(* IEC 61131-3 sources: generating_plc_code_with_llms/Code#1/ChatGPT_4/first run, 21 files *)

(* ---- 14.st ---- *)
// 41.85s
// 4
FUNCTION FC1001 : BOOL
VAR_INPUT
    MeasuredValue : REAL;  // The current measured value from the sensor
    SwitchValue   : REAL;  // The predetermined switch value
    Hysteresis    : REAL;  // The hysteresis in percentage of the switch value
END_VAR

VAR
    UpperLimit : REAL;
    LowerLimit : REAL;
END_VAR

// Calculate the upper and lower limits based on the hysteresis
UpperLimit := SwitchValue + (SwitchValue * Hysteresis / 100);
LowerLimit := SwitchValue - (SwitchValue * Hysteresis / 100);

// Logic to turn the output on or off based on the measured value and hysteresis
IF MeasuredValue > UpperLimit THEN
    FC1001 := TRUE;  // Turn on the output
ELSIF MeasuredValue < LowerLimit THEN
    FC1001 := FALSE; // Turn off the output
// If the value is within the hysteresis range, keep the output as is
END_IF

(* ---- 15.st ---- *)
// 58.63s
// 3
FUNCTION FC1002
VAR_INPUT
    SensorDetected : BOOL;  // TRUE if the ultrasonic sensor detects something
    E_A            : BOOL;  // The switch to turn the monitoring system on/off
END_VAR

VAR_OUTPUT
    P_HU           : BOOL;  // The horn for acoustic warning
    P_AL           : BOOL;  // The alarm
    P1             : BOOL;  // Indicator for monitoring system status
END_VAR

VAR
    DetectionTimer : TON;   // Timer for detection duration
END_VAR

// Turn on the monitoring system and indicate status
IF E_A THEN
    P1 := TRUE;
ELSE
    P1 := FALSE;
    P_HU := FALSE;  // Turn off horn when system is turned off
    P_AL := FALSE;  // Turn off alarm when system is turned off
END_IF

// Handling sensor detection
IF SensorDetected THEN
    IF NOT DetectionTimer.IN THEN
        DetectionTimer(IN := TRUE, PT := T#3s);  // Start timer when detection begins
    END_IF
    IF DetectionTimer.Q THEN
        P_HU := FALSE;  // Turn off horn after 3 seconds
        P_AL := TRUE;   // Turn on alarm after 3 seconds
    ELSE
        P_HU := TRUE;   // Turn on horn when detection is within 3 seconds
    END_IF
ELSE
    DetectionTimer(IN := FALSE);  // Reset timer when no detection
    P_HU := FALSE;                // Turn off horn if nothing is detected
    // Keep alarm on if it was already triggered, unless the system is turned off
END_IF

(* ---- 18.st ---- *)
// 37.97s
// 4
FUNCTION FC1003 : REAL
VAR_INPUT
    InputValue : REAL;    // The value from the sensor (0 to 255 in your case)
    IN_MIN     : REAL;    // Lower limit of the input range
    IN_MAX     : REAL;    // Upper limit of the input range
    OUT_MIN    : REAL;    // Lower limit of the output range (e.g., -20C)
    OUT_MAX    : REAL;    // Upper limit of the output range (e.g., 40C)
END_VAR

BEGIN
    // Linearly map the input value from its range to the output range
    FC1003 := OUT_MIN + (InputValue - IN_MIN) * (OUT_MAX - OUT_MIN) / (IN_MAX - IN_MIN);
END_FUNCTION

(* ---- 2.st ---- *)
//30.22s
//2
(* Function to calculate factorial *)
FUNCTION Factorial : LINT
VAR_INPUT
    n : UINT; (* non-negative integer *)
END_VAR
VAR
    result : LINT := 1; (* Initialize result to 1 *)
    i : UINT;
END_VAR

FOR i := 1 TO n DO
    result := result * LINT#(i);
END_FOR

Factorial := result;
END_FUNCTION

(* Function to calculate binomial coefficient *)
FUNCTION BinomialCoefficient : LINT
VAR_INPUT
    n : UINT; (* n in n choose k *)
    k : UINT; (* k in n choose k *)
END_VAR

IF k > n THEN
    RETURN 0; (* If k > n, then the coefficient is 0 *)
END_IF

BinomialCoefficient := Factorial(n) / (Factorial(k) * Factorial(n - k));
END_FUNCTION

(* ---- 3.st ---- *)
//20.48s
//2
FUNCTION Fibonacci : DINT
VAR_INPUT
    n : DINT; (* The index n for which the Fibonacci number is calculated *)
END_VAR
VAR
    a : DINT := 0;
    b : DINT := 1;
    temp : DINT;
    i : DINT;
END_VAR

IF n = 0 THEN
    RETURN 0;
ELSIF n = 1 THEN
    RETURN 1;
END_IF

FOR i := 2 TO n DO
    temp := a + b;
    a := b;
    b := temp;
END_FOR

Fibonacci := b;
END_FUNCTION

(* ---- 19.st ---- *)
// 56.28s
// 4
FUNCTION_BLOCK FB1005
VAR_INPUT
    START     : BOOL;    // Signal to start/stop measurement (from sensor S1)
    THICKNESS : DWORD;   // Measured thickness from lasers
    V_MAX     : REAL;    // Upper tolerance limit
    V_MIN     : REAL;    // Lower tolerance limit
END_VAR

VAR_OUTPUT
    M_MAX     : REAL;    // Maximum measured thickness
    M_MIN     : REAL;    // Minimum measured thickness
    P1        : BOOL;    // Reject light (ON if outside tolerance)
END_VAR

VAR
    CurrentThickness : REAL;
    MeasurementActive : BOOL;
END_VAR

BEGIN
    IF START THEN
        // Convert the DWORD thickness measurement to REAL
        CurrentThickness := DWORD_TO_REAL(THICKNESS);

        // Initialize min/max values at the start of a new measurement
        IF NOT MeasurementActive THEN
            M_MAX := CurrentThickness;
            M_MIN := CurrentThickness;
            MeasurementActive := TRUE;
        END_IF

        // Update min and max values
        IF CurrentThickness > M_MAX THEN
            M_MAX := CurrentThickness;
        END_IF
        IF CurrentThickness < M_MIN THEN
            M_MIN := CurrentThickness;
        END_IF
    ELSE
        // End of measurement, check tolerance and reset
        IF MeasurementActive THEN
            P1 := (M_MAX > V_MAX) OR (M_MIN < V_MIN);  // Check if outside tolerance
            MeasurementActive := FALSE;  // Reset for next cycle
        END_IF
    END_IF
END_FUNCTION_BLOCK

(* ---- 21.st ---- *)
// 108.14s
// 3
FUNCTION_BLOCK BURNER
VAR_INPUT
    IN           : BOOL;  // Start command
    OVER_TEMP    : BOOL;  // Boiler over-temperature protection
    OIL_TEMP     : BOOL;  // Oil reached temperature signal
    STAGE2       : BOOL;  // Command to activate stage 2
    MULTIPLE_IGNITION : BOOL; // Flag for retrying ignition
    RST          : BOOL;  // Reset command
END_VAR

VAR_OUTPUT
    PRE_HEAT     : BOOL;  // Pre-heating active
    FAIL         : BOOL;  // Failure state
    STATUS       : INT;   // Status code
END_VAR

VAR
    PRE_HEAT_TIME        : TON; // Timer for pre-heat time
    PRE_VENTILATION_TIME : TON; // Timer for pre-ventilation time
    PRE_IGNITE_TIME      : TON; // Timer before ignition
    SAFETY_TIME          : TON; // Timer for flame sensor safety check
    POST_IGNITE_TIME     : TON; // Timer for post-ignition operation
    STAGE2_DELAY         : TON; // Timer for delay to stage 2
    LOCKOUT_TIME         : TON; // Lockout timer after a fault
    OperationStage       : INT; // Current operation stage
    LockoutActive        : BOOL; // Lockout state
END_VAR

(* Additional implementation details would go here *)

(* ---- 1.st ---- *)
//29.01s
//4
PROGRAM AlarmControl
VAR
    xAlarm1 : BOOL; (* Variable for Alarm 1 *)
    xAlarm2 : BOOL; (* Variable for Alarm 2 *)
    xAllOn : BOOL; (* Signal to set all alarms on *)
    xAllOff : BOOL; (* Signal to set all alarms off *)
END_VAR

(* Turn on both alarms if xAllOn is activated *)
IF xAllOn THEN
    xAlarm1 := TRUE;
    xAlarm2 := TRUE;
    xAllOn := FALSE; (* Turn off the signal after setting alarms *)
END_IF

(* Turn off both alarms if xAllOff is activated *)
IF xAllOff THEN
    xAlarm1 := FALSE;
    xAlarm2 := FALSE;
    xAllOff := FALSE; (* Turn off the signal after resetting alarms *)
END_IF

END_PROGRAM

(* ---- 10.st ---- *)
//37.56s
//2
PROGRAM SigmoidFunction
VAR
    x : REAL; (* Input: the independent variable x *)
    sigmoid : REAL; (* Output: the value of the sigmoid function *)
    e : REAL; (* The base of natural logarithms *)
END_VAR

(* Set the value for the base of natural logarithms *)
e := 2.7182818284590452354; (* Approximate value of e *)

(* Calculate the sigmoid function *)
sigmoid := 1 / (1 + (e ** (-x)));

END_PROGRAM

(* ---- 11.st ---- *)
//30.17s
//4
PROGRAM SignFunction
VAR
    x : REAL; (* Input: the independent variable x *)
    sign : INT; (* Output: the value of the sign function *)
END_VAR

(* Calculate the sign function *)
IF x < 0 THEN
    sign := -1;
ELSIF x = 0 THEN
    sign := 0;
ELSE
    sign := 1;
END_IF;

END_PROGRAM

(* ---- 12.st ---- *)
//34.25s
//2
PROGRAM HyperbolicSineFunction
VAR
    x : REAL; (* Input: the independent variable x *)
    sinh_x : REAL; (* Output: the value of the hyperbolic sine function *)
    e : REAL; (* The base of natural logarithms *)
END_VAR

(* Set the value for the base of natural logarithms *)
e := 2.7182818284590452354; (* Approximate value of e *)

(* Calculate the hyperbolic sine function using the exponential function *)
sinh_x := (e ** x - e ** (-x)) / 2;

END_PROGRAM

(* ---- 13.st ---- *)
//48.01s
//2
PROGRAM NumberSearch
VAR
    numberList: ARRAY [1..100] OF INT; (* Array containing 100 random numbers *)
    found: BOOL; (* Output: TRUE if the number 10 is found, otherwise FALSE *)
    index: INT; (* Index for the current position in the list *)
END_VAR

(* Initialize variables *)
found := FALSE;
index := 1;

(* Search for the number 10 using REPEAT loop and EXIT statement *)
REPEAT
    IF numberList[index] = 10 THEN
        found := TRUE; (* Set found to TRUE if number 10 is found *)
        EXIT; (* Exit the loop *)
    END_IF;

    index := index + 1; (* Move to the next index *)
UNTIL index > 100; (* Exit the loop if the end of the list is reached *)

(* Output whether the number 10 was found *)
IF found THEN
    (* Implement actions to take if the number 10 is found *)
ELSE
    (* Implement actions to take if the number 10 is not found *)
END_IF;

END_PROGRAM

(* ---- 16.st ---- *)
//65.48s
//4
PROGRAM TrafficLightControl
VAR
    North_green, North_yellow, North_red: BOOL;
    East_green, East_yellow, East_red: BOOL;
    TrafficCycleTimer: TON;
END_VAR

(* Initialize the timer with PT as 10 seconds *)
TrafficCycleTimer(IN:= TRUE, PT:= T#10s);

(* Traffic light control logic *)
IF TrafficCycleTimer.ET < T#5s THEN
    North_green := TRUE;
    North_yellow := FALSE;
    North_red := FALSE;
    East_green := FALSE;
    East_yellow := FALSE;
    East_red := TRUE;
ELSIF TrafficCycleTimer.ET >= T#5s AND TrafficCycleTimer.ET < T#5500ms THEN
    North_green := FALSE;
    North_yellow := TRUE;
    North_red := FALSE;
    East_green := FALSE;
    East_yellow := FALSE;
    East_red := TRUE;
ELSIF TrafficCycleTimer.ET >= T#5500ms AND TrafficCycleTimer.ET < T#9500ms THEN
    North_green := FALSE;
    North_yellow := FALSE;
    North_red := TRUE;
    East_green := TRUE;
    East_yellow := FALSE;
    East_red := FALSE;
ELSIF TrafficCycleTimer.ET >= T#9500ms AND TrafficCycleTimer.ET < T#10s THEN
    North_green := FALSE;
    North_yellow := FALSE;
    North_red := TRUE;
    East_green := FALSE;
    East_yellow := TRUE;
    East_red := FALSE;
END_IF;

(* Reset the timer if the cycle is complete *)
IF TrafficCycleTimer.ET >= T#10s THEN
    TrafficCycleTimer.IN := FALSE; (* Stop the timer *)
    TrafficCycleTimer();           (* Reset the timer *)
    TrafficCycleTimer.IN := TRUE;  (* Restart the timer *)
END_IF;

TrafficCycleTimer(); (* Call the timer *)
END_PROGRAM

(* ---- 17.st ---- *)
//58.46s
//2
PROGRAM WeatherStation
VAR
    AnalogTempInput : INT; (* Input: Analog value representing the temperature *)
    AnalogHumidityInput : INT; (* Input: Analog value representing the humidity *)
    TemperatureC : REAL; (* The temperature in degrees Celsius *)
    Humidity : REAL; (* The humidity in percent *)
    DisplayText : STRING; (* Output: Text to display based on temperature and humidity *)
END_VAR

(* Constants for temperature conversion *)
CONST
    TEMP_SCALE : REAL := 0.1; (* Assuming the analog input represents temperature in tenths of degrees *)
    HUMIDITY_SCALE : REAL := 0.1; (* Assuming the analog input represents humidity in tenths of percent *)
END_CONST

(* Convert the analog inputs to meaningful values *)
TemperatureC := AnalogTempInput * TEMP_SCALE;
Humidity := AnalogHumidityInput * HUMIDITY_SCALE;

(* Evaluate temperature and humidity, then set display text *)
IF TemperatureC < 18 THEN
    DisplayText := 'Cold';
ELSIF TemperatureC <= 25 THEN
    (* Nested IF for humidity check within optimal temperature range *)
    IF Humidity >= 40 AND Humidity <= 75 THEN
        DisplayText := 'Opt';
    ELSE
        DisplayText := 'Temp. OK';
    END_IF;
ELSE
    DisplayText := 'Hot';
END_IF;

END_PROGRAM

(* ---- 20.st ---- *)
// 52.57s
// 4
PROGRAM InterlockProgram
VAR
    I1, I2      : BOOL;         // Inputs
    Q1, Q2      : BOOL;         // Outputs
    TL          : TIME;         // Dead time
    TimerQ1, TimerQ2 : TON;     // Timers for dead time
END_VAR

BEGIN
    // Update timers
    TimerQ1(IN := NOT Q1, PT := TL);
    TimerQ2(IN := NOT Q2, PT := TL);

    // Logic for Q1
    IF I1 AND TimerQ2.Q THEN
        Q1 := TRUE;
    ELSIF NOT I1 OR (I2 AND TimerQ1.Q) THEN
        Q1 := FALSE;
    END_IF

    // Logic for Q2
    IF I2 AND TimerQ1.Q THEN
        Q2 := TRUE;
    ELSIF NOT I2 OR (I1 AND TimerQ2.Q) THEN
        Q2 := FALSE;
    END_IF
END_PROGRAM

(* ---- 4.st ---- *)
//86.18s
//2
PROGRAM FillLevelCheck
VAR
    xAnalogValue : INT; (* Input: Fill level as analog value 0-32767 *)
    xFillLevelPercent : REAL; (* Converted fill level in percent *)
    xLowLevel : BOOL; (* Output: Low level indicator *)
    xOkLevel : BOOL; (* Output: OK level indicator *)
    xHighLevel : BOOL; (* Output: High level indicator *)
    xWarningHorn : BOOL; (* Output: Warning horn *)
END_VAR

(* Convert the analog value to a percentage: 0-32767 to 0-100% *)
xFillLevelPercent := (xAnalogValue / 32767) * 100;

(* Determine the fill level range using CASE instruction *)
CASE TRUE OF
    xFillLevelPercent < 1.0:
        xWarningHorn := TRUE; (* Activate warning horn *)
        xLowLevel := TRUE;
        xOkLevel := FALSE;
        xHighLevel := FALSE;
    xFillLevelPercent >= 1.0 AND xFillLevelPercent < 20.0:
        xLowLevel := TRUE; (* Indicate low level *)
        xOkLevel := FALSE;
        xHighLevel := FALSE;
        xWarningHorn := FALSE; (* Deactivate warning horn *)
    xFillLevelPercent >= 20.0 AND xFillLevelPercent < 80.0:
        xLowLevel := FALSE;
        xOkLevel := TRUE; (* Indicate OK level *)
        xHighLevel := FALSE;
        xWarningHorn := FALSE; (* Deactivate warning horn *)
    xFillLevelPercent >= 80.0:
        xLowLevel := FALSE;
        xOkLevel := FALSE;
        xHighLevel := TRUE; (* Indicate high level *)
        xWarningHorn := FALSE; (* Deactivate warning horn *)
END_CASE

END_PROGRAM

(* ---- 5.st ---- *)
//70.06s
//4
PROGRAM GateController
VAR
    Start_Loop : BOOL; (* Input: Control variable to start/stop the loop *)
    Gate_Open : BOOL; (* Output: Indicates if the gate is open *)
    One_Hour_Timer : TON; (* Timer that counts for 1 hour *)
    Sensor_Car : BOOL; (* Input: Senses the car *)
    Sensor_App : BOOL; (* Input: Senses the app *)
    Auth_Str : STRING; (* Input: Authorization string from the app or car *)
    my_defined_str : STRING := 'SecretPass'; (* Predefined authorization string *)
END_VAR

(* Initialize the timer with PT as 1 hour *)
One_Hour_Timer(PT := T#1h);

(* Start the one hour timer when Start_Loop is FALSE *)
IF NOT Start_Loop AND NOT One_Hour_Timer.Q THEN
    One_Hour_Timer.IN := TRUE; (* Start the timer *)
ELSIF Start_Loop OR One_Hour_Timer.Q THEN
    One_Hour_Timer.IN := FALSE; (* Stop the timer if Start_Loop is TRUE or the timer has finished *)
END_IF

(* Timer control logic *)
IF One_Hour_Timer.Q THEN
    IF Gate_Open THEN
        Gate_Open := FALSE; (* Close the gate if it's open after 1 hour *)
    END_IF
ELSE
    (* Check for car/app sensor and valid authorization string to open the gate *)
    IF (Sensor_Car OR Sensor_App) AND (Auth_Str = my_defined_str) THEN
        Gate_Open := TRUE; (* Open the gate if auth matches *)
    END_IF
END_IF

(* Update the timer *)
One_Hour_Timer();

END_PROGRAM

(* ---- 6.st ---- *)
//80.85s
//2
PROGRAM CraneLift
VAR
    doConvTop : BOOL; (* Output: Drives the top conveyor belt *)
    doConvBottom : BOOL; (* Output: Drives the bottom conveyor belt *)
    doConvLift : BOOL; (* Output: Drives the lift's conveyor belt *)
    doLiftTop : BOOL; (* Output: Moves the lift to the top position *)
    doLiftBottom : BOOL; (* Output: Moves the lift to the bottom position *)
    doLiftUnload : BOOL; (* Output: Moves the lift to the unloading position *)
    diConvTop : BOOL; (* Input: Light barrier for the top conveyor belt *)
    diConvBottom : BOOL; (* Input: Light barrier for the bottom conveyor belt *)
    diLiftTop : BOOL; (* Input: Sensor indicating the lift is at the top position *)
    diLiftBottom : BOOL; (* Input: Sensor indicating the lift is at the bottom position *)
    diLiftUnload : BOOL; (* Input: Sensor indicating the lift is at the unloading position *)
    diBoxLift : BOOL; (* Input: Sensor indicating the box is completely at the lift *)
    LiftRequested : BOOL; (* Internal: Indicates if the lift has been requested *)
    LiftPosition : STRING := ''; (* Internal: Indicates the requested position of the lift *)
END_VAR

(* Check light barriers and request lift *)
IF diConvTop THEN
    doConvTop := FALSE; (* Stop top conveyor belt *)
    LiftRequested := TRUE;
    LiftPosition := 'Top';
ELSIF diConvBottom THEN
    doConvBottom := FALSE; (* Stop bottom conveyor belt *)
    LiftRequested := TRUE;
    LiftPosition := 'Bottom';
END_IF

(* Move lift to requested position if not already there *)
IF LiftRequested THEN
    CASE LiftPosition OF
        'Top':
            IF NOT diLiftTop THEN
                doLiftTop := TRUE; (* Move lift to top *)
                doLiftBottom := FALSE;
                doLiftUnload := FALSE;
            END_IF
        'Bottom':
            IF NOT diLiftBottom THEN
                doLiftBottom := TRUE; (* Move lift to bottom *)
                doLiftTop := FALSE;
                doLiftUnload := FALSE;
            END_IF
    END_CASE
END_IF

(* When lift is in position and the box is completely at the lift, move to unloading *)
IF (LiftPosition = 'Top' AND diLiftTop) OR (LiftPosition = 'Bottom' AND diLiftBottom) THEN
    IF diBoxLift THEN
        doConvLift := TRUE; (* Turn on lift conveyor belt *)
        IF diLiftUnload THEN
            (* When crate is at unloading position, unload the crate *)
            doLiftUnload := TRUE;
            doConvTop := FALSE;
            doConvBottom := FALSE;
            doConvLift := FALSE;
            LiftRequested := FALSE; (* Reset lift request *)
        END_IF
    END_IF
END_IF

END_PROGRAM

(* ---- 7.st ---- *)
//54.32s
//2
(* Define constants *)
CONST
    NUM_RECEPTORS : INT := 5; (* Number of load receptors *)
    MAX_VALUE : INT := 32767; (* Maximum value for each receptor *)
END_CONST

PROGRAM CraneLoadCalculation
VAR
    aiLoadReceptor1 : INT; (* Analog input value from load receptor 1 *)
    aiLoadReceptor2 : INT; (* Analog input value from load receptor 2 *)
    aiLoadReceptor3 : INT; (* Analog input value from load receptor 3 *)
    aiLoadReceptor4 : INT; (* Analog input value from load receptor 4 *)
    aiLoadReceptor5 : INT; (* Analog input value from load receptor 5 *)
    TotalLoad : INT; (* Sum of loads from all receptors *)
    AverageLoad : REAL; (* Average load across receptors *)
END_VAR

VAR CONSTANT
    MAX_ANALOG_VALUE : INT := MAX_VALUE; (* Replace fixed max value *)
    TOTAL_RECEPTORS : INT := NUM_RECEPTORS; (* Replace fixed count *)
END_VAR

TotalLoad := 0; (* Initialize TotalLoad *)
AverageLoad := 0; (* Initialize AverageLoad *)

(* Sum the loads from all receptors using a FOR loop *)
FOR i := 1 TO TOTAL_RECEPTORS DO
    CASE i OF
        1:
            TotalLoad := TotalLoad + aiLoadReceptor1;
        2:
            TotalLoad := TotalLoad + aiLoadReceptor2;
        3:
            TotalLoad := TotalLoad + aiLoadReceptor3;
        4:
            TotalLoad := TotalLoad + aiLoadReceptor4;
        5:
            TotalLoad := TotalLoad + aiLoadReceptor5;
    END_CASE
END_FOR

(* Calculate the average load *)
AverageLoad := TotalLoad / REAL(TOTAL_RECEPTORS);

END_PROGRAM

(* ---- 8.st ---- *)
//32.92s
//2
PROGRAM LambertWFunction
VAR
    x : REAL; (* Input: the value for which we want to compute the Lambert W function *)
    w : REAL; (* Output: the approximation of the Lambert W function *)
    tol : REAL; (* Tolerance for the approximation *)
    max_iter : INT; (* Maximum number of iterations *)
    iter : INT; (* Iterator *)
    e : REAL; (* Base of natural logarithm *)
    w_next : REAL; (* Next approximation of the Lambert W function *)
END_VAR

(* Initialize variables *)
w := 0; (* Initial guess for W(x) *)
tol := 1E-5; (* Set the tolerance for the approximation *)
max_iter := 100; (* Set the maximum number of iterations *)
iter := 0; (* Initialize iteration counter *)
e := 2.71828182845904523536; (* Approximation of e *)

(* Implementing Halley's method to approximate the Lambert W function *)
REPEAT
    w_next := w - ((w * e ** w - x) / (e ** w + w * e ** (2 * w)));
    iter := iter + 1;
    IF ABS(w_next - w) < tol OR iter >= max_iter THEN
        EXIT;
    END_IF;
    w := w_next;
UNTIL FALSE;

(* Output the result *)
w := w_next;

END_PROGRAM

(* ---- 9.st ---- *)
//31.7s
//4
PROGRAM LeapYearCheck
VAR
    YEAR : INT; (* Input: Year to check *)
    IsLeapYear : BOOL; (* Output: TRUE if YEAR is a leap year, otherwise FALSE *)
END_VAR

(* A year is a leap year if it is divisible by 4 but not by 100, unless it is also divisible by 400 *)
IsLeapYear := (YEAR MOD 4 = 0) AND ((YEAR MOD 100 <> 0) OR (YEAR MOD 400 = 0));

END_PROGRAM
